ADAPTER IMode (* Adapter Interface *)
  (* Standard: 61499-1 *)
  (* Version 0.0, 11/16/2023, SESA371406, Schneider Electric *)
  PACKAGE SE.Nereda;
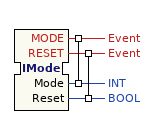
  EVENT_OUTPUT
    MODE WITH Mode; (* Response from Socket *)
    RESET WITH Reset; (* Request from Socket *)
  END_EVENT
  VAR_OUTPUT
    Mode : INT; (* Response Data from Socket *)
    Reset : BOOL; (* Request Data from Socket *)
  END_VAR
  SERVICE SOCKET/PLUG
    SEQUENCE request_confirm
      SOCKET.RESET(Reset) -> PLUG.RESET(Reset);
      PLUG.CNF(CNFD) -> SOCKET.CNF(CNFD);
    END_SEQUENCE
    SEQUENCE indication_response
      PLUG.IND(INDD) -> SOCKET.IND(INDD);
      SOCKET.MODE(Mode) -> PLUG.MODE(Mode);
    END_SEQUENCE
  END_SERVICE
END_ADAPTER
